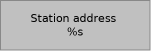
VISUALIZATION _VisuAddressShow  // 151x51
    Rectangle (1,1 148x48), "Station address %s", text variable: ComGVL._glAddressNameTable[ComGVL._glAddressSelectionIndex]
END_VISUALIZATION

(* stored: Version 1.1.0.1, ProductVersion 3.1.4024.2
   Visu _VisuAddressShow: Id {c5536179-8e52-4788-9063-ed1dfbfcc7bd} *)
